// TIA Portal V21 export
VAR_GLOBAL   // PLC tag table "K_Passo_Produzione_SterilizzatoreTubo"
END_VAR
VAR_GLOBAL CONSTANT   // user constants
   K_Passo_Sterilizzazione : Int := 1;
   K_Passo_Riempimento : Int := 2;
   K_Passo_Lavoro : Int := 3;
   K_Passo_Svuotamento : Int := 4;
   K_Passo_RisciacquoFineSvuotamento : Int := 5;
END_VAR
